(* IEC 61131-3 sources: BODAS-HelloWorld/extracted_st/bodas_rc18_12_40/plc_logic/application/01_maintask/03_communication/00_can/function/func_can1rxdatabox1_cbk, 1 file *)

(* ---- FUNC_CAN1RxDatabox1_Cbk.st ---- *)
(* --- Interface --- *)
(*********************************************************************************************************************
 *     __   __   ___  ___           __   __        __   __  ___
 *   /_ / /  / /__  /    /__/     /_ / /_   |_ / /_ / /  /  /  /__/
 *  /__/ /__/ __ / /__  /  /     /  | /__  /  | /  | /__/  /  /  /
 *
 * Project: Hello World for ml290.rts
 *
 * FUNC: FUNC_CAN1RxDatabox1_Cbk
 *
 * Author:
 *
 * Description:
 * Callback for CAN1
 *
 * (c) Copyright by BOSCH REXROTH AG, all rights reserved
 *
 *********************************************************************************************************************)
FUNCTION FUNC_CAN1RxDatabox1_Cbk
VAR
END_VAR

(* --- Implementation --- *)
GlobalVariables.can1RxDataboxCbkCntr_gu32 := GlobalVariables.can1RxDataboxCbkCntr_gu32 + 1;
